(* CODESYS project Ladder1.project

Project tree, tasks and I/O mapping:
  Device : CODESYS Control Win V3, 3S - Smart Software Solutions GmbH, version 3.5.15.30
    application Application
      libraries: Standard, * (System)
      task MainTask (cyclic, interval t#20ms, priority 1) calls PLC_PRG
      task VISU_TASK (cyclic, interval 100 ms, priority 31) calls VisuElems.Visu_Prg
      program PLC_PRG [LD]
      visualisation Visualization
  text list GlobalTextList
*)

// Device/Application/PLC_PRG
PROGRAM PLC_PRG
VAR
	Contact1: BOOL;
	Coil1: BOOL;
	Contact2: BOOL := FALSE;
END_VAR

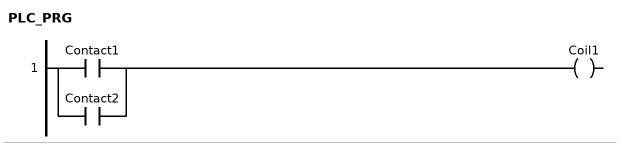
// NETWORK 1
Coil1 := Contact1 OR Contact2;

END_PROGRAM

// Device/Application/Visualization
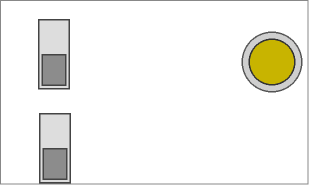
VISUALIZATION Visualization  // 309x185
    DipSwitch (19,19 70x70), variable: PLC_PRG.Contact1, behaviour: TOGGLE, style: Switch-DipSwitch-Gray
    Lamp1 (237,27 70x70), variable: PLC_PRG.Coil1, style: Lamp-Lamp1-Yellow
    DipSwitch (20,113 70x70), variable: PLC_PRG.Contact2, behaviour: TOGGLE, style: Switch-DipSwitch-Gray
END_VISUALIZATION
